FUNCTION_BLOCK Stage15 (* Template for a Basic Function Block Type *)
  (* Standard: 61499-2 *)
  (* Version 1.0, 2021-06-20, HP *)
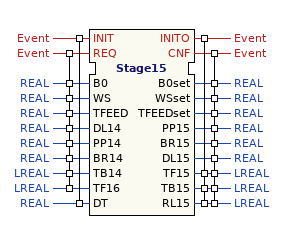
  EVENT_INPUT
    INIT WITH DT; (* Initialization Request *)
    REQ WITH B0, WS, TFEED, DL14, PP14, BR14, TB14, TF16; (* Normal Execution Request *)
  END_EVENT
  EVENT_OUTPUT
    INITO WITH TB15, TF15, RL15; (* Initialization Confirm *)
    CNF WITH TB15, DL15, TF15, BR15, PP15, RL15, TFEEDset, WSset, B0set; (* Execution Confirmation *)
  END_EVENT
  VAR_INPUT
    B0 : REAL;
    WS : REAL;
    TFEED : REAL;
    DL14 : REAL;
    PP14 : REAL;
    BR14 : REAL;
    TB14 : LREAL;
    TF16 : LREAL;
    DT : REAL;
  END_VAR
  VAR_OUTPUT
    B0set : REAL;
    WSset : REAL;
    TFEEDset : REAL;
    PP15 : REAL;
    BR15 : REAL;
    DL15 : REAL;
    TF15 : LREAL;
    TB15 : LREAL;
    RL15 : LREAL;
  END_VAR
  VAR
    AB : REAL; (* internal variabel *)
    UU : REAL;
    TREF : REAL;
    AD : REAL;
    AHC : REAL;
    AHR : REAL;
    AS : REAL;
    REC : REAL;
    WN : REAL;
    WN_1 : REAL;
    XKN : REAL;
    C1 : REAL;
    HS : REAL;
    G : REAL;
    W1 : REAL;
    TFREC : REAL;
    TS : REAL;
    DTS : REAL;
    TF15_last : REAL;
    RL15_last : REAL;
    TB15_last : REAL;
    USS : REAL;
    RHOB : REAL;
    CPB : REAL;
    CPF : REAL;
    FMW : REAL;
    HLV : REAL;
    HV : REAL;
    BPR : REAL;
    FMC : REAL;
    U : REAL;
    A : REAL;
    B : REAL;
    C : REAL;
    D1 : REAL;
    d : REAL;
    a : REAL;
    A1 : REAL;
    A2 : REAL;
    A3 : REAL;
    A4 : REAL;
    A5 : REAL;
    A6 : REAL;
    p : REAL;
    q : REAL;
    TC : REAL;
    PC : REAL;
    DTB15 : REAL;
    DEN15 : REAL;
    DH15 : REAL;
    DP15 : REAL;
    DPDH15 : REAL;
    DT15 : REAL;
    m : REAL;
    n : REAL;
    VR15 : REAL;
    DELTA15 : REAL;
    DELTA37 : REAL;
    DELTA59 : REAL;
    DELTA15_last : REAL;
    DELTA37_last : REAL;
    DELTA59_last : REAL;
  END_VAR
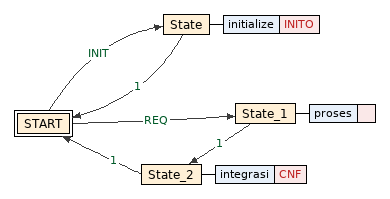
  EC_STATES
    START; (* Initial State *)
    State : initialize -> INITO;
    State_1 : proses;
    State_2 : integrasi -> CNF;
  END_STATES
  EC_TRANSITIONS
    START TO State := INIT;
    State TO START := 1;
    START TO State_1 := REQ;
    State_1 TO State_2 := 1;
    State_2 TO START := 1;
  END_TRANSITIONS
  ALGORITHM initialize IN ST: (* Initialization algorithm *)
TREF :=273.15;
AB :=57.2727;
AHC :=4069.2;
AHR :=2639.7;
AS :=3225.7;
REC :=0.0;
//TF2:=TF2;

//TFEED :=TFEED1+TREF;
 //TS:=TS1+TREF;
WN :=3.0;
XKN :=0.68;
HS:=0.11;
G :=9.81;
W1 :=0.50;

RL15 := 0.604150913563253;
TB15 := 328.045077472691;
TF15 := 324.575567486082;
TF16 := 322.379704977734;


RL15_last :=RL15;
TB15_last :=TB15;
TF15_last :=TF15;
  END_ALGORITHM
  ALGORITHM proses IN ST: (* kalkulasi *)
UU := TFEED;
U :=UU;

USS :=49.767;
C1 :=0.625;
RHOB :=1032.4; //maassa jenis brine
CPB :=1.00; //heatcapacity Brine
CPF :=1.00; //heat capacity feed
FMW :=23654.0;
HLV :=563.7959;
HV :=625.1971;
BPR :=2.192;
FMC :=34736.09;
//U :=UU; //feed temp



///  Calculate the physical properties

//A :=3.2437814;
//B :=5.86826*0.001;
//C :=1.1702379*0.00000001;
//D1 :=2.1878462*0.001;
//TC :=647.27;
//PC :=218.167;


A1 :=3.2437814;
A2:=5.86826*0.001;
A3:=1.1702379*0.00000001;
A4 :=2.1878462*0.001;
A5 :=647.27;
A6 :=218.167;

DTB15 :=A5-TB15;
DEN15 :=(A1+A2*DTB15+A3*DTB15*DTB15*DTB15)/(1+A4*DTB15)*DTB15/TB15;
p:=DEN15;
q:=10.0;
PP15 :=A6/(EXPT(q, p));

// calculate the brine flow rates
DP15:=PP14-PP15;
DH15:=RL15-C1*HS;
DPDH15 :=DP15*101000+G*RHOB*DH15;
m:=DPDH15*RHOB;
n:=0.5;
BR15 :=WN*XKN*RL15*(EXPT(m, n));
BR15 :=BR15*60.0/1000.0;

// calculate the vapor flow rates

DT15 :=TB15-BPR/1.8-(TF16+TF15)*0.5;
VR15:=U*AHC*DT15/HLV/1000.0;
DL15 :=DL14+VR15;


//// state equation
DELTA15 :=(BR14-BR15-VR15)*1000.0/RHOB/AB;
DELTA37 :=((BR14*CPB*(TB14-TB15))-VR15*(HV-CPB*(TB15-TREF)))*1000.0/AB/RHOB/CPB/RL15;
DELTA59 :=(B0*CPF*(TF16-TF15)*1000+(U*AHC*DT15))/FMW/CPF;
  END_ALGORITHM
  ALGORITHM integrasi IN ST: (* new algorithm *)
B0set:=B0;
WSset:=WS ;
TFEEDset:=TFEED;
//integrasi
RL15 := (DELTA15 + DELTA15_last)*0.5*DT + RL15_last;
DELTA15_last :=DELTA15 ;
RL15_last :=RL15;

TB15:= (DELTA37 + DELTA37_last)*0.5*DT + TB15_last;
DELTA37_last :=DELTA37 ;
TB15_last:=TB15;

TF15 := (DELTA59 + DELTA59_last)*0.5*DT + TF15_last;
DELTA59_last :=DELTA59 ;
TF15_last :=TF15;
  END_ALGORITHM
END_FUNCTION_BLOCK
